PROGRAM F18_ClearSystemQueues
VAR
	fbClearHMIQueue			: FB_SYSTEM_ClearHMIQueue;

	fbClearMasterListArray	: FB_SYSTEM_ClearMasterListArray;
	fbClearPackArray		: FB_SYSTEM_ClearPackArray;
	fbClearOuterArray		: FB_SYSTEM_ClearOuterArray;
	fbClearCasePackerArray 	: FB_SYSTEM_ClearCasePackerArray;
	fbClearCaseDataArray	: FB_SYSTEM_ClearCaseDataArray;

	fbClearCameraStatus		: FB_SYSTEM_ClearCameraStatus;

	ftEnablePrimaryMasterList		: F_TRIG;
	ftEnableSecondaryMasterList	: F_TRIG;

	rtClearMasterListWithOpenStatus			: R_TRIG;
	rtClearAggregationWithOpenStatus			: R_TRIG;
	rtClearStackerQueueWithOpenStatus			: R_TRIG;
	rtClearInterimQueueWithOpenStatus			: R_TRIG;

	tofTPDConditionalOFFDelay 		: TOF;

	tofDoneTimer			: TOF;

END_VAR

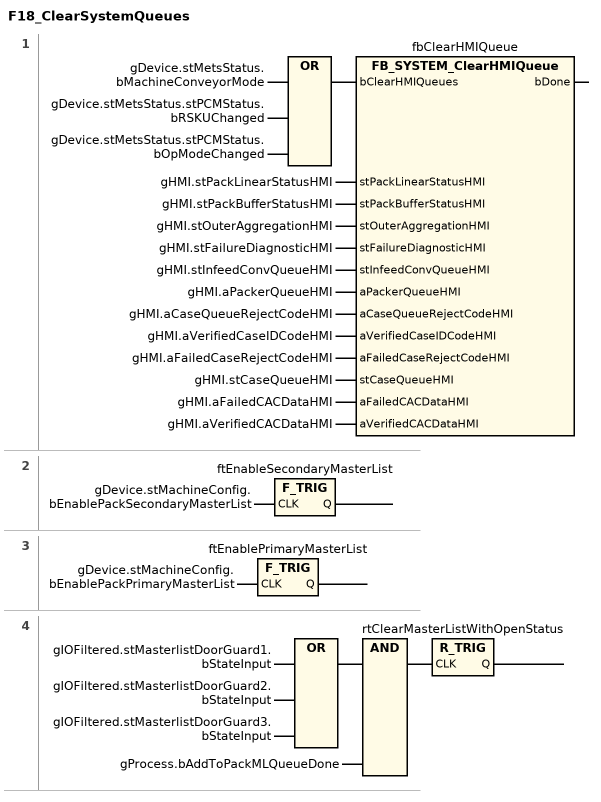
// NETWORK 1
fbClearHMIQueue(
    bClearHMIQueues := gDevice.stMetsStatus.bMachineConveyorMode OR gDevice.stMetsStatus.stPCMStatus.bRSKUChanged OR gDevice.stMetsStatus.stPCMStatus.bOpModeChanged,
    stPackLinearStatusHMI := gHMI.stPackLinearStatusHMI,
    stPackBufferStatusHMI := gHMI.stPackBufferStatusHMI,
    stOuterAggregationHMI := gHMI.stOuterAggregationHMI,
    stFailureDiagnosticHMI := gHMI.stFailureDiagnosticHMI,
    stInfeedConvQueueHMI := gHMI.stInfeedConvQueueHMI,
    aPackerQueueHMI := gHMI.aPackerQueueHMI,
    aCaseQueueRejectCodeHMI := gHMI.aCaseQueueRejectCodeHMI,
    aVerifiedCaseIDCodeHMI := gHMI.aVerifiedCaseIDCodeHMI,
    aFailedCaseRejectCodeHMI := gHMI.aFailedCaseRejectCodeHMI,
    stCaseQueueHMI := gHMI.stCaseQueueHMI,
    aFailedCACDataHMI := gHMI.aFailedCACDataHMI,
    aVerifiedCACDataHMI := gHMI.aVerifiedCACDataHMI); // FB_SYSTEM_ClearHMIQueue

// NETWORK 2
ftEnableSecondaryMasterList(CLK := gDevice.stMachineConfig.bEnablePackSecondaryMasterList); // F_TRIG

// NETWORK 3
ftEnablePrimaryMasterList(CLK := gDevice.stMachineConfig.bEnablePackPrimaryMasterList); // F_TRIG

// NETWORK 4
rtClearMasterListWithOpenStatus(CLK := (gIOFiltered.stMasterlistDoorGuard1.bStateInput OR gIOFiltered.stMasterlistDoorGuard2.bStateInput OR gIOFiltered.stMasterlistDoorGuard3.bStateInput) AND gProcess.bAddToPackMLQueueDone); // R_TRIG

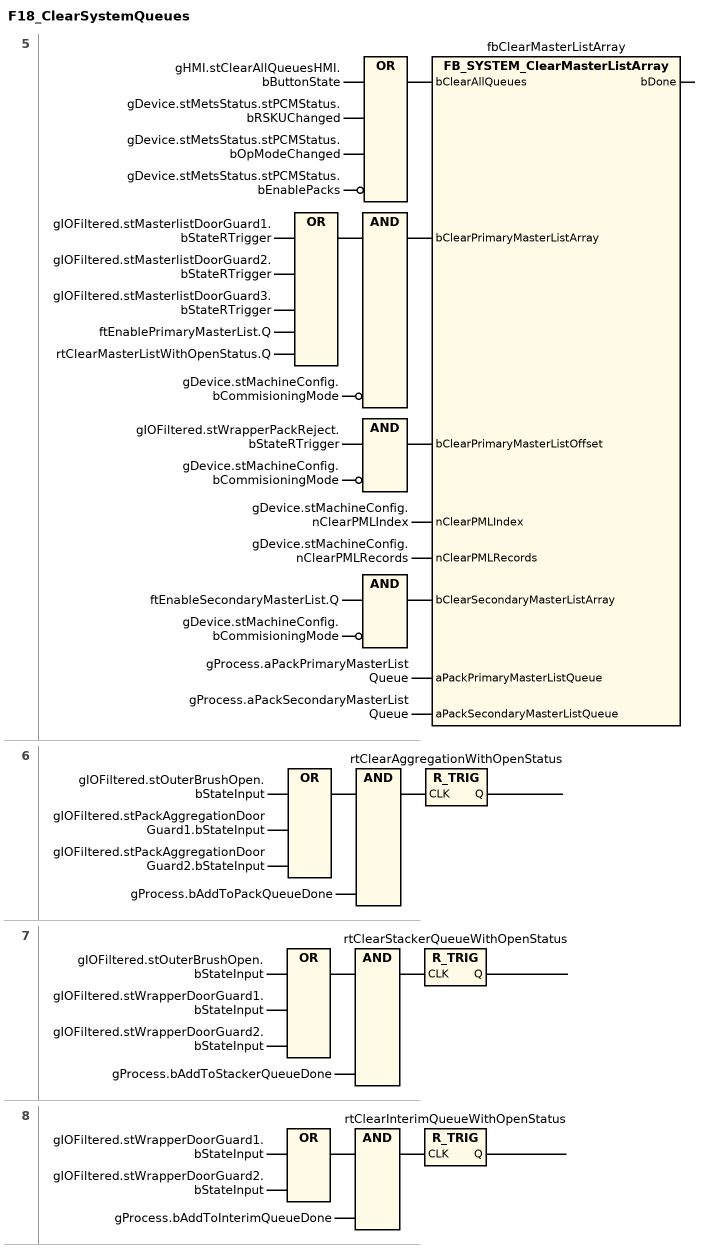
// NETWORK 5
fbClearMasterListArray(
    bClearAllQueues := gHMI.stClearAllQueuesHMI.bButtonState OR gDevice.stMetsStatus.stPCMStatus.bRSKUChanged OR gDevice.stMetsStatus.stPCMStatus.bOpModeChanged OR NOT gDevice.stMetsStatus.stPCMStatus.bEnablePacks,
    bClearPrimaryMasterListArray := (gIOFiltered.stMasterlistDoorGuard1.bStateRTrigger OR gIOFiltered.stMasterlistDoorGuard2.bStateRTrigger OR gIOFiltered.stMasterlistDoorGuard3.bStateRTrigger OR ftEnablePrimaryMasterList.Q OR rtClearMasterListWithOpenStatus.Q) AND NOT gDevice.stMachineConfig.bCommisioningMode,
    bClearPrimaryMasterListOffset := gIOFiltered.stWrapperPackReject.bStateRTrigger AND NOT gDevice.stMachineConfig.bCommisioningMode,
    nClearPMLIndex := gDevice.stMachineConfig.nClearPMLIndex,
    nClearPMLRecords := gDevice.stMachineConfig.nClearPMLRecords,
    bClearSecondaryMasterListArray := ftEnableSecondaryMasterList.Q AND NOT gDevice.stMachineConfig.bCommisioningMode,
    aPackPrimaryMasterListQueue := gProcess.aPackPrimaryMasterListQueue,
    aPackSecondaryMasterListQueue := gProcess.aPackSecondaryMasterListQueue); // FB_SYSTEM_ClearMasterListArray

// NETWORK 6
rtClearAggregationWithOpenStatus(CLK := (gIOFiltered.stOuterBrushOpen.bStateInput OR gIOFiltered.stPackAggregationDoorGuard1.bStateInput OR gIOFiltered.stPackAggregationDoorGuard2.bStateInput) AND gProcess.bAddToPackQueueDone); // R_TRIG

// NETWORK 7
rtClearStackerQueueWithOpenStatus(CLK := (gIOFiltered.stOuterBrushOpen.bStateInput OR gIOFiltered.stWrapperDoorGuard1.bStateInput OR gIOFiltered.stWrapperDoorGuard2.bStateInput) AND gProcess.bAddToStackerQueueDone); // R_TRIG

// NETWORK 8
rtClearInterimQueueWithOpenStatus(CLK := (gIOFiltered.stWrapperDoorGuard1.bStateInput OR gIOFiltered.stWrapperDoorGuard2.bStateInput) AND gProcess.bAddToInterimQueueDone); // R_TRIG

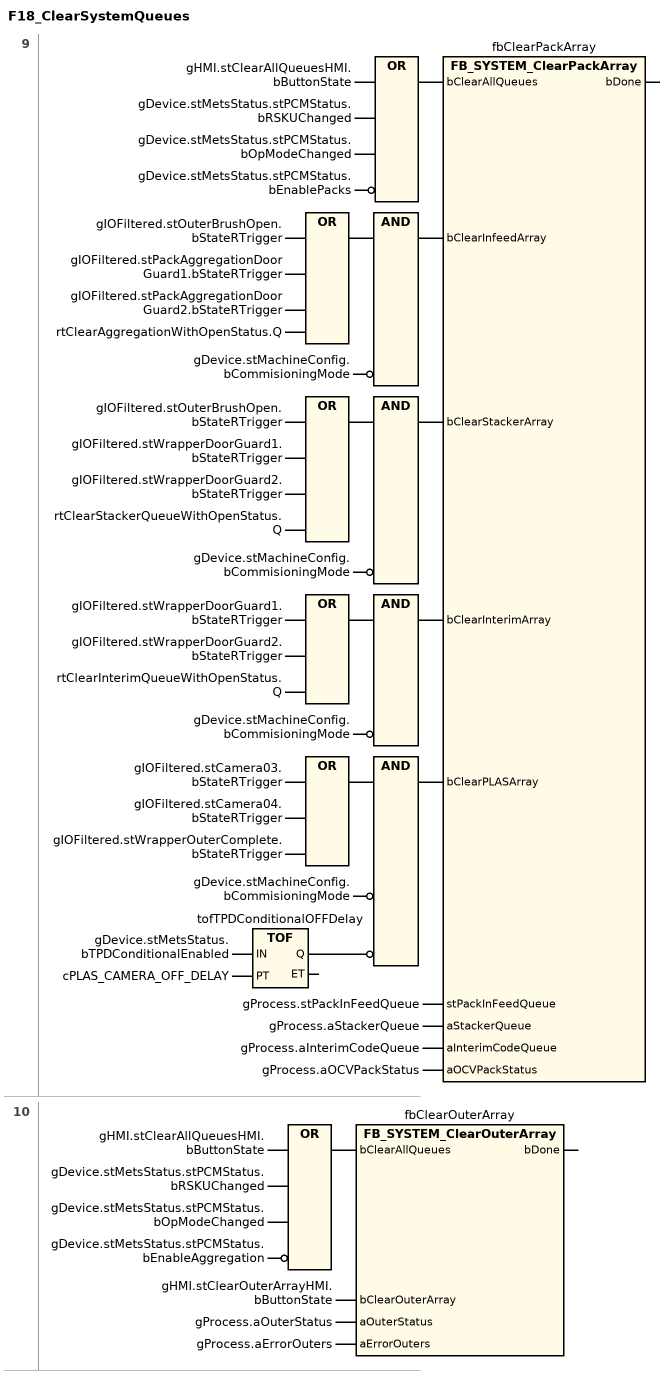
// NETWORK 9
tofTPDConditionalOFFDelay(IN := gDevice.stMetsStatus.bTPDConditionalEnabled, PT := cPLAS_CAMERA_OFF_DELAY); // TOF
fbClearPackArray(
    bClearAllQueues := gHMI.stClearAllQueuesHMI.bButtonState OR gDevice.stMetsStatus.stPCMStatus.bRSKUChanged OR gDevice.stMetsStatus.stPCMStatus.bOpModeChanged OR NOT gDevice.stMetsStatus.stPCMStatus.bEnablePacks,
    bClearInfeedArray := (gIOFiltered.stOuterBrushOpen.bStateRTrigger OR gIOFiltered.stPackAggregationDoorGuard1.bStateRTrigger OR gIOFiltered.stPackAggregationDoorGuard2.bStateRTrigger OR rtClearAggregationWithOpenStatus.Q) AND NOT gDevice.stMachineConfig.bCommisioningMode,
    bClearStackerArray := (gIOFiltered.stOuterBrushOpen.bStateRTrigger OR gIOFiltered.stWrapperDoorGuard1.bStateRTrigger OR gIOFiltered.stWrapperDoorGuard2.bStateRTrigger OR rtClearStackerQueueWithOpenStatus.Q) AND NOT gDevice.stMachineConfig.bCommisioningMode,
    bClearInterimArray := (gIOFiltered.stWrapperDoorGuard1.bStateRTrigger OR gIOFiltered.stWrapperDoorGuard2.bStateRTrigger OR rtClearInterimQueueWithOpenStatus.Q) AND NOT gDevice.stMachineConfig.bCommisioningMode,
    bClearPLASArray := (gIOFiltered.stCamera03.bStateRTrigger OR gIOFiltered.stCamera04.bStateRTrigger OR gIOFiltered.stWrapperOuterComplete.bStateRTrigger) AND NOT gDevice.stMachineConfig.bCommisioningMode AND NOT tofTPDConditionalOFFDelay.Q,
    stPackInFeedQueue := gProcess.stPackInFeedQueue,
    aStackerQueue := gProcess.aStackerQueue,
    aInterimCodeQueue := gProcess.aInterimCodeQueue,
    aOCVPackStatus := gProcess.aOCVPackStatus); // FB_SYSTEM_ClearPackArray

// NETWORK 10
fbClearOuterArray(
    bClearAllQueues := gHMI.stClearAllQueuesHMI.bButtonState OR gDevice.stMetsStatus.stPCMStatus.bRSKUChanged OR gDevice.stMetsStatus.stPCMStatus.bOpModeChanged OR NOT gDevice.stMetsStatus.stPCMStatus.bEnableAggregation,
    bClearOuterArray := gHMI.stClearOuterArrayHMI.bButtonState,
    aOuterStatus := gProcess.aOuterStatus,
    aErrorOuters := gProcess.aErrorOuters); // FB_SYSTEM_ClearOuterArray

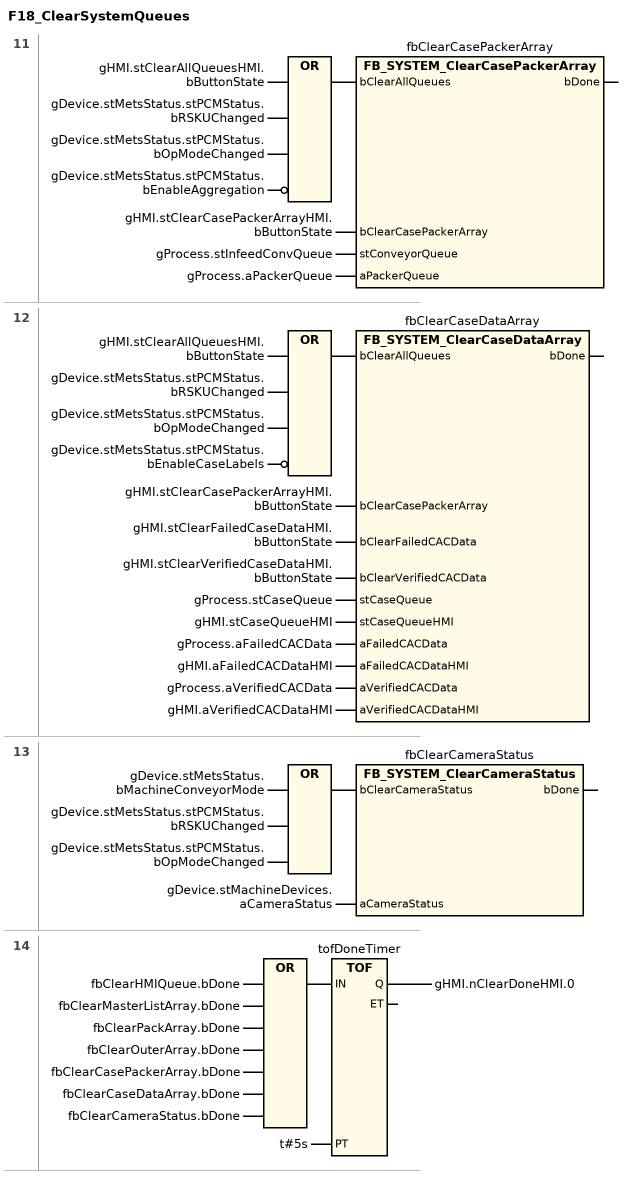
// NETWORK 11
fbClearCasePackerArray(
    bClearAllQueues := gHMI.stClearAllQueuesHMI.bButtonState OR gDevice.stMetsStatus.stPCMStatus.bRSKUChanged OR gDevice.stMetsStatus.stPCMStatus.bOpModeChanged OR NOT gDevice.stMetsStatus.stPCMStatus.bEnableAggregation,
    bClearCasePackerArray := gHMI.stClearCasePackerArrayHMI.bButtonState,
    stConveyorQueue := gProcess.stInfeedConvQueue,
    aPackerQueue := gProcess.aPackerQueue); // FB_SYSTEM_ClearCasePackerArray

// NETWORK 12
fbClearCaseDataArray(
    bClearAllQueues := gHMI.stClearAllQueuesHMI.bButtonState OR gDevice.stMetsStatus.stPCMStatus.bRSKUChanged OR gDevice.stMetsStatus.stPCMStatus.bOpModeChanged OR NOT gDevice.stMetsStatus.stPCMStatus.bEnableCaseLabels,
    bClearCasePackerArray := gHMI.stClearCasePackerArrayHMI.bButtonState,
    bClearFailedCACData := gHMI.stClearFailedCaseDataHMI.bButtonState,
    bClearVerifiedCACData := gHMI.stClearVerifiedCaseDataHMI.bButtonState,
    stCaseQueue := gProcess.stCaseQueue,
    stCaseQueueHMI := gHMI.stCaseQueueHMI,
    aFailedCACData := gProcess.aFailedCACData,
    aFailedCACDataHMI := gHMI.aFailedCACDataHMI,
    aVerifiedCACData := gProcess.aVerifiedCACData,
    aVerifiedCACDataHMI := gHMI.aVerifiedCACDataHMI); // FB_SYSTEM_ClearCaseDataArray

// NETWORK 13
fbClearCameraStatus(bClearCameraStatus := gDevice.stMetsStatus.bMachineConveyorMode OR gDevice.stMetsStatus.stPCMStatus.bRSKUChanged OR gDevice.stMetsStatus.stPCMStatus.bOpModeChanged, aCameraStatus := gDevice.stMachineDevices.aCameraStatus); // FB_SYSTEM_ClearCameraStatus

// NETWORK 14
tofDoneTimer(IN := fbClearHMIQueue.bDone OR fbClearMasterListArray.bDone OR fbClearPackArray.bDone OR fbClearOuterArray.bDone OR fbClearCasePackerArray.bDone OR fbClearCaseDataArray.bDone OR fbClearCameraStatus.bDone, PT := t#5s); // TOF
gHMI.nClearDoneHMI.0 := tofDoneTimer.Q;

END_PROGRAM

(* stored: Version 1.1.0.1
   POU F18_ClearSystemQueues: Id {fa972d2f-43ca-476e-86b3-087c8b0d3a06}, SpecialFunc None *)
